Staubli VAL3: RobotController.dtx

mdesc mNomSpeed
public string sMotionTaskName
public string sScreenTaskName
public string sDataTaskName
public string sExceptTaskName
public string sCommTaskName
public string sMotionSocket
public string sFbkSocket
public FlagStatus fFlagStatus
  [0]
    num ForceFlag
    num RosFlag
    num RobotFlag
